FUNCTION_BLOCK passforward
  (* Standard: 61499-2 *)
  (* Version 0.1, 2017-00-09, Hammond, HAMMONDSDESKTOP *)
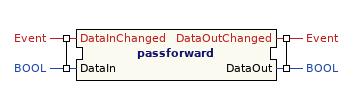
  EVENT_INPUT
    DataInChanged WITH DataIn;
  END_EVENT
  EVENT_OUTPUT
    DataOutChanged WITH DataOut;
  END_EVENT
  VAR_INPUT
    DataIn : BOOL;
  END_VAR
  VAR_OUTPUT
    DataOut : BOOL;
  END_VAR
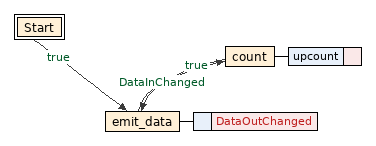
  EC_STATES
    Start;
    emit_data : -> DataOutChanged;
    count : upcount;
  END_STATES
  EC_TRANSITIONS
    Start TO emit_data := true;
    emit_data TO count := DataInChanged;
    count TO emit_data := true;
  END_TRANSITIONS
  ALGORITHM upcount IN C:
printf("Received %i\n", me->DataIn);
me->DataOut = me->DataIn + 1;
  END_ALGORITHM
END_FUNCTION_BLOCK
